// TIA Portal V16 export
// export: Created 2021-07-12T14:47:18.721626Z, ExportSetting WithDefaults, DisplayName Totally Integrated Automation Portal, DisplayVersion V16, DisplayName TIA Portal Version Control Interface, DisplayVersion V16, DisplayName TIA Portal Openness, DisplayVersion V16, DisplayName STEP 7 Professional, DisplayVersion V16, DisplayName STEP 7 Safety, DisplayVersion V16, DisplayName WinCC Professional, DisplayVersion V16
TYPE "LSimaHydTO_typeStatusForceProfile"
TITLE = LSimaHydTO_typeStatusForceProfile
// Indicates the status of a force profile processing
// stored: IsFailsafeCompliant false
   STRUCT
      ActualProfile : UInt := 0;   // Currently effective force profile DB number
      ForceProfileMode : DInt := 0;   // 0: with force value / 1: profile is a function of time / 2: profile is a function of position
      Active : Bool := FALSE;   // Activation status of a command for specifying the force profile
      State : DInt := 0;   // Execution state: 0: inactive / 1: in interpolation / 2: on profile / 3: profile end
      BaseValue : LReal := 0.0;   // Current reference value
      ProfileValue : LReal := 0.0;   // Profile value for the base value
   END_STRUCT;
END_TYPE
